(* CODESYS project opc_ua_server_on_raspi.project

Project tree, tasks and I/O mapping:
  RaspiSPS : CODESYS Control for Raspberry Pi, 3S - Smart Software Solutions GmbH, version 3.5.11.20
    application Application
      libraries: Standard, * (System)
      task MainTask (cyclic, interval 4 ms, priority 1) calls PLC_PRG
      program PLC_PRG [CFC]
      Symbols
    SoftMotion General Axis Pool
    I²C
    SPI
    GPIOs_A_B : GPIOs A/B, 3S - Smart Software Solutions GmbH, version 3.5.11.0
        unmapped channels: digital inputs (GPIO0..GPIO31), digital outputs (GPIO0..GPIO31)
    Onewire
    Camera device
      <Leer>
*)

// RaspiSPS/Application/PLC_PRG
PROGRAM PLC_PRG
VAR
	eingang1: BOOL;
	eingang2: BOOL;
	ausgang: BOOL;
END_VAR

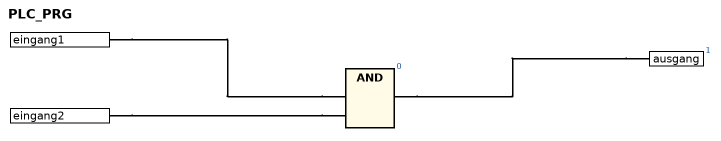
ausgang := eingang1 AND eingang2;

END_PROGRAM
